FUNCTION_BLOCK FB_RawToAnalog
VAR_INPUT
	iRaw: INT;
	iBits: UINT;
	fMax: LREAL;
	fMin: LREAL;
END_VAR
VAR_OUTPUT
	fReal: LREAL;
END_VAR
VAR
	fScale: LREAL;
END_VAR

// Converts the integer from an analog input terminal to a real unit value (e.g., volts)
IF fScale = 0 AND fMax > fMin THEN
	fScale := (EXPT(2, iBits) - 1) / (fMax - fMin);
END_IF
IF fScale <> 0 THEN
	fReal := iRaw / fScale + fMin;
END_IF

END_FUNCTION_BLOCK

(* stored: Version 1.1.0.1, ProductVersion 3.1.4022.12
   POU FB_RawToAnalog: Id {98817c2d-2670-42a6-be0a-6b1209bb15af}, SpecialFunc None *)
